Fanuc TP program (LS listing): SET_UFRAME_TP.ls

/PROG  SET_UFRAME_TP
/ATTR
OWNER		= MNEDITOR;
COMMENT		= "SET UFRAME NUM";
PROG_SIZE	= 152;
CREATE		= DATE 25-10-10  TIME 14:00:00;
MODIFIED	= DATE 25-10-10  TIME 14:00:00;
FILE_NAME	= ;
VERSION		= 0;
LINE_COUNT	= 1;
MEMORY_SIZE	= 520;
PROTECT		= READ_WRITE;
TCD:  STACK_SIZE	= 0,
      TASK_PRIORITY	= 50,
      TIME_SLICE	= 0,
      BUSY_LAMP_OFF	= 0,
      ABORT_REQUEST	= 0,
      PAUSE_REQUEST	= 0;
DEFAULT_GROUP	= 1,*,*,*,*;
CONTROL_CODE	= 00000000 00000000;
/APPL
/MN
   1:  UFRAME_NUM = R[85:FANUC_REMOTE_USER_NUM] ;
/POS
/END
